// TIA Portal V20 export
TYPE "LKinCtrl_typeCOffReturn"
   STRUCT
      returnValue : Word;   // Return value
      region : Int;   // Region type - see LKinCtrl_OffsetContour
      subBlockNumber : DInt;   // Sub function block number
      internalNumber : DInt;   // Internal number indicates the source code position
   END_STRUCT;
END_TYPE
